ABB RobotStudio station: Tema3_FINAL.rspag

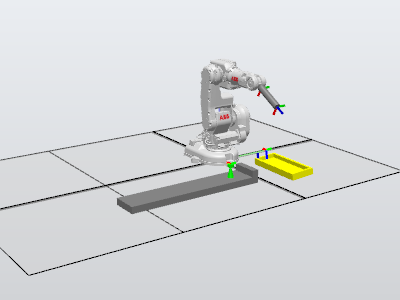
--- station ---
Station Tema2 (saved by RobotStudio 23.2.10478.1)
Controller IRB140_6_81
  mechanical unit ROB_1: IRB140_6_81_C_03, 6 joints, base frame (0, 0, 0) mm
Layout (positions relative to the parent item):
  - IRB140_6_81_C_03 [mechanism, from %ABB.RobotStudio.Models.IRB140%\IRB140_6_81_C_G_03.rslib] at (0, 0, 0) mm; joint values [0, 0, 0, 0, 0.5236, 0] (rad or m)
  - Piesa_1 [part, from Components\Piesa.rslib] at (472.23, -240.64, 150) mm, rotated rx 180 ry 0 rz 180 deg
  - Cutie_depunere [part] at (490.45, 242.38, 41.53) mm, rotated rx 1.86 ry 5.61 rz -94.5 deg, size 185.7 x 485.7 x 50 mm
  - MyNewTool [mechanism] at (506.29, 0, 679.5) mm, rotated rx 180 ry 60 rz 180 deg
      TCP MyNewTool at (0, 0, 200) mm
      links: Part_1
  - Source [smart component, from Components\Source.rslib]
      properties: Source=Piesa_1; Copy=(none); Parent=(none); Position=[0.472235 -0.240636 0.15]; Orientation=[3.14159265358979 1.22460635382238E-16 -3.14159265358979]; Transient=false; PhysicsBehavior=-1
  - Queue [smart component, from Components\Queue.rslib]
      properties: Back=(none); Front=(none); Queue=; NumberOfObjects=0
  - Banda [part] at (368.51, -1112.89, 0) mm, size 200 x 1000 x 50 mm
  - Stop [part] at (368.68, -113.43, 0) mm, size 200 x 50 x 100 mm
Attachment: MyNewTool is attached to IRB140_6_81_C_03 / Link6
EventTableEntry 2296: ActivationMode=2, Cyclic=false, Group=, Trigger=aa_gripper 2297, Actions=[EventTableActionAttach 2298], Comment=
EventTableTriggerIO 2297: Operator=0, IOValue=[1], IRC5Controller=? -1, SignalSource=IRB140_6_81 1186
EventTableActionAttach 2298: MountObject=true, FlangeIndext=0, FindNearest=true, AttachmentParent=MyNewTool 2307, AttachmentChild=? -1, Offset=[X=1, Y=0, Z=0, W=0, X=0, Y=1, Z=0, W=0, X=0, Y=0, Z=1, W=0, X=0, Y=0, Z=0, W=1]
EventTableEntry 2311: ActivationMode=2, Cyclic=false, Group=, Trigger=aa_gripper 2312, Actions=[EventTableActionDetach 2313], Comment=
EventTableTriggerIO 2312: Operator=0, IOValue=[0], IRC5Controller=? -1, SignalSource=IRB140_6_81 1186
EventTableActionDetach 2313: AttachmentParent=MyNewTool 2307, AttachmentChild=? -1
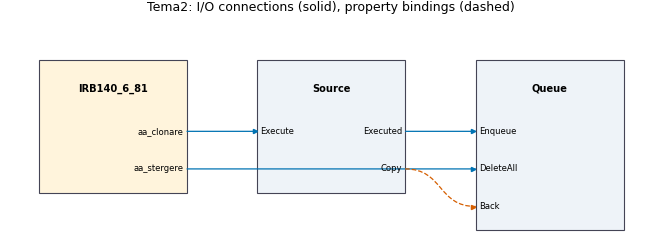
Station logic (signal -> signal, property => property):
  IRB140_6_81.aa_clonare -> Source.Execute
  Source.Executed -> Queue.Enqueue
  IRB140_6_81.aa_stergere -> Queue.DeleteAll
  Source.Copy => Queue.Back

--- Controller Data/IRB140_6_81/RAPID/TASK1/PROGMOD/CalibData.mod ---
MODULE CalibData
    PERS tooldata MyNewTool:=[TRUE,[[0,0,200],[1,0,0,0]],[1,[0,0,1],[1,0,0,0],0,0,0]];
    TASK PERS wobjdata plan_inclinat:=[FALSE,TRUE,"",[[262.764,188.299,27.226],[0.997872,0.0482292,-0.0180937,-0.0399847]],[[0,0,0],[1,0,0,0]]];
ENDMODULE

--- Controller Data/IRB140_6_81/RAPID/TASK1/PROGMOD/Module1.mod ---
MODULE Module1
        CONST robtarget home:=[[679.496732003,0,579.5],[0.5,0,0.866025404,0],[0,0,0,0],[9E+09,9E+09,9E+09,9E+09,9E+09,9E+09]];
    CONST robtarget P_pick:=[[472.235,-240.636,150],[0,0,1,0],[-1,0,-1,0],[9E+09,9E+09,9E+09,9E+09,9E+09,9E+09]];
    CONST robtarget P_place:=[[55.327278058,44.868249435,100],[0,0,1,0],[0,0,0,0],[9E+09,9E+09,9E+09,9E+09,9E+09,9E+09]];
    VAR robtarget my_pick;
    VAR robtarget my_place;
!***********************************************************
    !
    ! Module:  Module1
    !
    ! Description:
    !   <Insert description here>
    !
    ! Author: Lenovo
    !
    ! Version: 1.0
    !
    !***********************************************************


    !***********************************************************
    !
    ! Procedure main
    !
    !   This is the entry point of your program
    !
    !***********************************************************
    PROC main()
        !Add your code here

        MoveJ home,v1000,z100,MyNewTool\WObj:=wobj0;
        my_pick:=P_pick;
        SetDO aa_clonare,0;
        SetDO aa_stergere,0;
        FOR i FROM 0 TO 23 DO
            SetDO aa_clonare,1;
            my_place:=offs(P_place,(i mod 6)*60,((i div 6) mod 2)*60,100*(i div 12));
            pick_and_place;
            SetDO aa_clonare,0;
        ENDFOR

      !  FOR i FROM 12 TO 23 DO
      !      my_pick:=offs(P_pick,(i mod 3)*70,((i div 3) mod 4)*70,-100);
      !      my_place:=offs(P_place,(i mod 6)*60,((i div 6) mod 2)*60,+100);
      !  ENDFOR
        MoveL home,v1000,z100,MyNewTool\WObj:=wobj0;
        SetDO aa_stergere,1;
        MoveL P_pick,v1000,z100,MyNewTool\WObj:=wobj0;
    ENDPROC

    PROC pick_and_place()
        SetDO aa_gripper, 0;
        !MoveJ home,v1000,z100,MyNewTool\WObj:=wobj0;

        MoveJ offs(my_pick,0,0,200),v1000,fine,MyNewTool\WObj:=wobj0;
        MoveL my_pick,v1000,fine,MyNewTool\WObj:=wobj0;
        SetDO aa_gripper,1;
        !WaitTime 0.5;
        MoveL offs(my_pick,0,0,250),v1000,fine,MyNewTool\WObj:=wobj0;

        MoveJ offs(my_place,0,0,250),v1000,fine,MyNewTool\WObj:=plan_inclinat;
        MoveL my_place,v1000,fine,MyNewTool\WObj:=plan_inclinat;
        SetDO aa_gripper,0;
        !WaitTime 0.5;
        MoveL offs(my_place,0,0,200),v1000,fine,MyNewTool\WObj:=plan_inclinat;

        !MoveJ home,v1000,z100,MyNewTool\WObj:=wobj0;
    ENDPROC
ENDMODULE

--- Controller Data/IRB140_6_81/SYSPAR/EIO.cfg ---
EIO:CFG_1.0:6:1::
#
EIO_SIGNAL:

      -Name "aa_gripper" -SignalType "DO" -Access "All"

      -Name "aa_clonare" -SignalType "DO" -Access "All"

      -Name "aa_stergere" -SignalType "DO" -Access "All"
